PROGRAM CraneSimulation
VAR
	fTime : LREAL;
	fOilLevelSensor : LREAL;
	eOilLevelAlarms : DUT_oil_level;
	fCraneAngle : LREAL;
	fCraneAngleDeg : LREAL;
END_VAR

IF inputs.bAutoMode AND inputs.bStart THEN
	fTime := fTime + parameters.pCraneParameters.fCycleTime;
ELSE
	fTime := 0;
END_IF

IF fTime > 0 AND inputs.bAutoMode THEN
	outputs.bSimRunning := TRUE;
END_IF
IF outputs.bSimRunning THEN
	IF fTime > 0 AND fTime <= parameters.pCraneParameters.fT2 THEN
		outputs.fCylinderVelocity := 1/(parameters.pCraneParameters.fT2);
		outputs.fCylinderPosition := outputs.fCylinderVelocity*fTime;
		parameters.pCraneParameters.fMidPos := outputs.fCylinderPosition;//saved for next loop
	ELSIF fTime > parameters.pCraneParameters.fT2 AND fTime <= parameters.pCraneParameters.fT3 THEN
		outputs.fCylinderVelocity := -1/(parameters.pCraneParameters.fT3-Parameters.pCraneParameters.fT2);
		outputs.fCylinderPosition := outputs.fCylinderVelocity*(fTime-parameters.pCraneParameters.fT2) + parameters.pCraneParameters.fMidPos;
	ELSE
		outputs.fCylinderVelocity := 0;
	END_IF

//	outputs.fCylinderVelocity := inputs.fCylinderVelocityReference;
//	outputs.fCylinderPosition := 0.5*outputs.fCylinderVelocity*fTime*fTime + parameters.fInitialVelocity*fTime + parameters.fInitialPosition;
END_IF


IF inputs.bReset THEN
	fTime := 0;
	inputs.bStart := FALSE;
	inputs.bEnable := FALSE;
	inputs.bReset := FALSE;
	outputs.fCylinderPosition := parameters.pCraneParameters.fInitialPosition;
	outputs.fCylinderVelocity := parameters.pCraneParameters.fInitialVelocity;
END_IF
//oil level
IF fOilLevelSensor < 20 THEN
	eOilLevelAlarms := DUT_oil_level.VeryLow;
	ELSIF fOilLevelSensor > 200 THEN
		eOilLevelAlarms := DUT_oil_level.VeryHigh;
	ELSE
		eOilLevelAlarms := DUT_oil_level.OK;		
END_IF
fCraneAngle := F_degToRad(fDeg := fCraneAngleDeg);

END_PROGRAM

(* stored: Version 1.1.0.1, ProductVersion 3.1.4024.10
   POU CraneSimulation: Id {386eb2ba-0859-427d-9c1c-15458717297f}, SpecialFunc None *)
